FUNCTION CelsiusToFahrenheit  : REAL
VAR_INPUT
	TemperatureInCelsius :REAL;
END_VAR
VAR
	Temp:REAL;
END_VAR

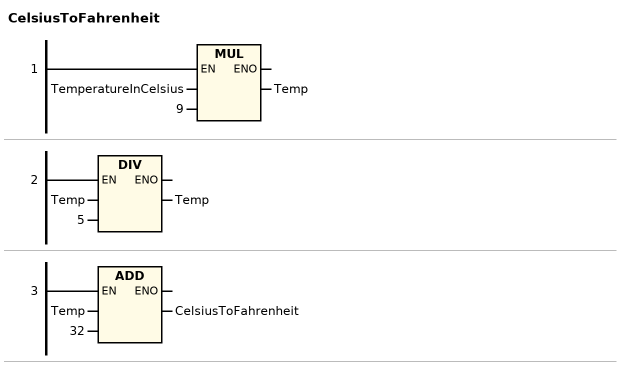
// NETWORK 1
Temp := TemperatureInCelsius * 9;

// NETWORK 2
Temp := Temp / 5;

// NETWORK 3
CelsiusToFahrenheit := Temp + 32;

END_FUNCTION

(* stored: Version 1.1.0.1, ProductVersion 3.1.4020.12
   POU CelsiusToFahrenheit: Id {37bc4548-f547-4137-b2f7-dfc6ba521d37}, SpecialFunc None *)
